FUNCTION_BLOCK FrequencyMeasurement EXTENDS SM_FrequencyMeasurement
VAR_INPUT
END_VAR
VAR_OUTPUT
END_VAR
VAR
    noOfSamples : UINT := 100;
    _toStatus : MeasurementToStatus;
	_executeMovingAverage : BOOL;
    _ctrl_moving_avg : FB_CTRL_MOVING_AVERAGE;
    _params : ST_CTRL_MOVING_AVERAGE_PARAMS;
    _array : ARRAY [1..100] OF LREAL;
END_VAR

SUPER^(config := config);

_params.nSamplesToFilter  := noOfSamples;
_params.tCtrlCycleTime    := GLOBAL.config.PLC_CTRL_TIME;

// only call the _ctrl_moving_avg FB once per task cycle (not once every time the xxxMeasurement FB is called)
IF _executeMovingAverage <> GLOBAL.config.PLC_TASK_FLIP THEN
	_executeMovingAverage := GLOBAL.config.PLC_TASK_FLIP;
	_ctrl_moving_avg(
		fIn             := actual.hertz.value,
		fManSyncValue   := 0.0,
		bSync           := FALSE,
		eMode           := E_CTRL_MODE.eCTRL_MODE_ACTIVE,
		bHold           := FALSE,
		stParams        := _params);
END_IF

// update the average value
average(newHertzValue := _ctrl_moving_avg.fOut);
	
_toStatus(
    overrange     := overrange,
    underrange    := underrange,
    error         := error,
    alarmStatus   := statuses.alarmStatus,
    enabledStatus := statuses.enabledStatus,
    actualStatus  => actualStatus);
	
SUPER^(config := config);

METHOD FB_init : BOOL
VAR_INPUT
	bInitRetains : BOOL; // if TRUE, the retain variables are initialized (warm start / cold start)
	bInCopyCode : BOOL;  // if TRUE, the instance afterwards gets moved into the copy code (online change)
END_VAR
_params.tTaskCycleTime    := GLOBAL.config.PLC_TASK_TIME;
_params.pWorkArray_ADR    := ADR(_array);
_params.nWorkArray_SIZEOF := SIZEOF(_array);
END_METHOD

END_FUNCTION_BLOCK

(* stored: Version 1.1.0.1, ProductVersion 3.1.4018.5
   POU FrequencyMeasurement: Id {9e0b9b1a-10c2-4646-af61-17aa4ac58258}, SpecialFunc None
   Method FB_init: Id {6dcfaec3-32d4-4529-a5b9-186ddf5c1008} *)
